PROGRAM MAIN
VAR
    fbDiffBPTest    :    FB_DiffBP_Test;
    fbBPTMTest    :    FB_BPTM_Test;
    //fbSafeBPCompareTest    :    FB_SafeBPCompare_Test;
    //fbevWithinSpecTest    :    FB_evWithinSpec_Test;
    //fbPEWTest    :    FB_PhotonEnergyWatcher_Test;
    fbFFTest    :    FB_FastFault_Test;
    fbArbiterTest    :    FB_Arbiter_Test;
    //fbevRangeCalcTest : FB_evRangeCalculator_Test;
    fbSubSysToArbTest : FB_SubsysToArb_Test;
    fbArbToSubSysTest : FB_ArbToSubsys_Test;
END_VAR

TcUnit.RUN();

END_PROGRAM

(* stored: Version 1.1.0.1, ProductVersion 3.1.4022.18
   POU MAIN: Id {87d6bba0-cac0-4c5b-b8ef-b01bdb9ad7f6}, SpecialFunc None *)
